(* IEC 61131-3 sources: LStream-JSON-XML/test, 4 files *)

(* ---- JsonDeserializerTests.st ---- *)
USING Simatic.Ax;
USING AxUnit;
USING Simatic.Ax.LStream;
USING Simatic.Ax.LStream.Utilities;
USING Simatic.Ax.System.Strings;
using Simatic.Ax.LStream.Models;

NAMESPACE LStreamTest

    ///////////////// Tests for JSON Blocks
    {TestFixture}
    CLASS JsonDeserializerTests
        VAR
            //Test1 (Test to try the LStream_JsonDeserializer.st by deserializing a JSON (inputString1 & inputString2) and comparing its output with the expected tree (expectedTreeOutput1))
            jsonDeserializer : LStream_JsonDeserializer;
            inputString1 : STRING := '{"sessionContext": {"sessionId": "154237171615905","locale": "en_US","persId": 0},"methodName": "valeo2WC.cfWipClose","inArgs": [{"mode": "0","stationNumber": "SubRib0101","step": "0010","cycleTime": "253.2","unitArray": [';
            inputString2 : STRING := '{"unit": "HLF659734","pos": "1", "state": "1","failArray": [{"failCode": "Condensator position","compName": "BOMPOS60"}]},{"unit": "HLF659735","pos": "2", "state": "0"}]}]}';
            rawInput1 : ARRAY[0..10000] OF BYTE;
            actualTreeOutput : ARRAY[0..200] OF LStream_typeElement;
            expectedTreeOutput1 : ARRAY[0..200] OF LStream_typeElement;

            //Test2 (Test to try the LStream_JsonDeserializer.st when the input JSON has empty brackets as value in the key (In this example: "items":[] & "edges":[]). The deserialize output tree is compared with the expected tree (expectedTreeOutput2))
            jsonDeserializer2 : LStream_JsonDeserializer;
            inputString3 : STRING := '{"id":"A","nodes":[{"nodeId":"CAT","items":[],"sequenceId":"A","released":"WORD","nodePosition":{"x":"1"}}],"edges":[]}';
            rawInput2 : ARRAY[0..10000] OF BYTE;
            actualTreeOutput2 : ARRAY[0..200] OF LStream_typeElement;
            expectedTreeOutput2 : ARRAY[0..200] OF LStream_typeElement;

       END_VAR

        {FixtureSetup}
        METHOD PUBLIC TestSetup

            //Test1 Setup
            StringToByteArray(string1 := inputString1, string2 := inputString2, byteArray := rawInput1);

            expectedTreeOutput1[0].types := SINT#16#0;
            expectedTreeOutput1[0].key := 'sessionContext';
            expectedTreeOutput1[0].value := 'NULL';
            expectedTreeOutput1[0].depth := SINT#16#0;
            expectedTreeOutput1[0].closingElement := FALSE;

            expectedTreeOutput1[1].types := SINT#16#02;
            expectedTreeOutput1[1].key := 'sessionId';
            expectedTreeOutput1[1].value := '154237171615905';
            expectedTreeOutput1[1].depth := SINT#16#01;
            expectedTreeOutput1[1].closingElement := FALSE;

            expectedTreeOutput1[2].types := SINT#16#02;
            expectedTreeOutput1[2].key := 'locale';
            expectedTreeOutput1[2].value := 'en_US';
            expectedTreeOutput1[2].depth := SINT#16#01;
            expectedTreeOutput1[2].closingElement := FALSE;

            expectedTreeOutput1[3].types := SINT#16#03;
            expectedTreeOutput1[3].key := 'persId';
            expectedTreeOutput1[3].value := '0';
            expectedTreeOutput1[3].depth := SINT#16#01;
            expectedTreeOutput1[3].closingElement := TRUE;

            expectedTreeOutput1[4].types := SINT#16#02;
            expectedTreeOutput1[4].key := 'methodName';
            expectedTreeOutput1[4].value := 'valeo2WC.cfWipClose';
            expectedTreeOutput1[4].depth := SINT#16#0;
            expectedTreeOutput1[4].closingElement := FALSE;

            expectedTreeOutput1[5].types := SINT#16#01;
            expectedTreeOutput1[5].key := 'inArgs';
            expectedTreeOutput1[5].value := 'NULL';
            expectedTreeOutput1[5].depth := SINT#16#0;
            expectedTreeOutput1[5].closingElement := false;

            expectedTreeOutput1[6].types := SINT#16#02;
            expectedTreeOutput1[6].key := 'mode';
            expectedTreeOutput1[6].value := '0';
            expectedTreeOutput1[6].depth := SINT#16#02;
            expectedTreeOutput1[6].closingElement := false;

            expectedTreeOutput1[7].types := SINT#16#02;
            expectedTreeOutput1[7].key := 'stationNumber';
            expectedTreeOutput1[7].value := 'SubRib0101';
            expectedTreeOutput1[7].depth := SINT#16#02;
            expectedTreeOutput1[7].closingElement := false;

            expectedTreeOutput1[8].types := SINT#16#02;
            expectedTreeOutput1[8].key := 'step';
            expectedTreeOutput1[8].value := '0010';
            expectedTreeOutput1[8].depth := SINT#16#02;
            expectedTreeOutput1[8].closingElement := false;

            expectedTreeOutput1[9].types := SINT#16#02;
            expectedTreeOutput1[9].key := 'cycleTime';
            expectedTreeOutput1[9].value := '253.2';
            expectedTreeOutput1[9].depth := SINT#16#02;
            expectedTreeOutput1[9].closingElement := false;

            expectedTreeOutput1[10].types := SINT#16#01;
            expectedTreeOutput1[10].key := 'unitArray';
            expectedTreeOutput1[10].value := 'NULL';
            expectedTreeOutput1[10].depth := SINT#16#02;
            expectedTreeOutput1[10].closingElement := false;

            expectedTreeOutput1[11].types := SINT#16#02;
            expectedTreeOutput1[11].key := 'unit';
            expectedTreeOutput1[11].value := 'HLF659734';
            expectedTreeOutput1[11].depth := SINT#16#04;
            expectedTreeOutput1[11].closingElement := false;

            expectedTreeOutput1[12].types := SINT#16#02;
            expectedTreeOutput1[12].key := 'pos';
            expectedTreeOutput1[12].value := '1';
            expectedTreeOutput1[12].depth := SINT#16#04;
            expectedTreeOutput1[12].closingElement := false;

            expectedTreeOutput1[13].types := SINT#16#02;
            expectedTreeOutput1[13].key := 'state';
            expectedTreeOutput1[13].value := '1';
            expectedTreeOutput1[13].depth := SINT#16#04;
            expectedTreeOutput1[13].closingElement := false;

            expectedTreeOutput1[14].types := SINT#16#01;
            expectedTreeOutput1[14].key := 'failArray';
            expectedTreeOutput1[14].value := 'NULL';
            expectedTreeOutput1[14].depth := SINT#16#04;
            expectedTreeOutput1[14].closingElement := false;

            expectedTreeOutput1[15].types := SINT#16#02;
            expectedTreeOutput1[15].key := 'failCode';
            expectedTreeOutput1[15].value := 'Condensator position';
            expectedTreeOutput1[15].depth := SINT#16#06;
            expectedTreeOutput1[15].closingElement := false;

            expectedTreeOutput1[16].types := SINT#16#02;
            expectedTreeOutput1[16].key := 'compName';
            expectedTreeOutput1[16].value := 'BOMPOS60';
            expectedTreeOutput1[16].depth := SINT#16#06;
            expectedTreeOutput1[16].closingElement := true;

            expectedTreeOutput1[17].types := SINT#16#02;
            expectedTreeOutput1[17].key := 'unit';
            expectedTreeOutput1[17].value := 'HLF659735';
            expectedTreeOutput1[17].depth := SINT#16#04;
            expectedTreeOutput1[17].closingElement := FALSE;

            expectedTreeOutput1[18].types := SINT#16#02;
            expectedTreeOutput1[18].key := 'pos';
            expectedTreeOutput1[18].value := '2';
            expectedTreeOutput1[18].depth := SINT#16#04;
            expectedTreeOutput1[18].closingElement := FALSE;

            expectedTreeOutput1[19].types := SINT#16#02;
            expectedTreeOutput1[19].key := 'state';
            expectedTreeOutput1[19].value := '0';
            expectedTreeOutput1[19].depth := SINT#16#04;
            expectedTreeOutput1[19].closingElement := true;

            //Test Setup Json Deserializer case 2
            StringToByteArray(string1 := inputString3, byteArray := rawInput2);

            expectedTreeOutput2[0].types := SINT#16#02;
            expectedTreeOutput2[0].key := 'id';
            expectedTreeOutput2[0].value := 'A';
            expectedTreeOutput2[0].depth := SINT#16#0;
            expectedTreeOutput2[0].closingElement := FALSE;

            expectedTreeOutput2[1].types := SINT#16#01;
            expectedTreeOutput2[1].key := 'nodes';
            expectedTreeOutput2[1].value := 'NULL';
            expectedTreeOutput2[1].depth := SINT#16#0;
            expectedTreeOutput2[1].closingElement := FALSE;

            expectedTreeOutput2[2].types := SINT#16#02;
            expectedTreeOutput2[2].key := 'nodeId';
            expectedTreeOutput2[2].value := 'CAT';
            expectedTreeOutput2[2].depth := SINT#16#02;
            expectedTreeOutput2[2].closingElement := FALSE;

            expectedTreeOutput2[3].types := SINT#16#01;
            expectedTreeOutput2[3].key := 'items';
            expectedTreeOutput2[3].value := 'NULL';
            expectedTreeOutput2[3].depth := SINT#16#02;
            expectedTreeOutput2[3].closingElement := FALSE;

            expectedTreeOutput2[4].types := SINT#16#02;
            expectedTreeOutput2[4].key := 'sequenceId';
            expectedTreeOutput2[4].value := 'A';
            expectedTreeOutput2[4].depth := SINT#16#02;
            expectedTreeOutput2[4].closingElement := FALSE;

            expectedTreeOutput2[5].types := SINT#16#02;
            expectedTreeOutput2[5].key := 'released';
            expectedTreeOutput2[5].value := 'WORD';
            expectedTreeOutput2[5].depth := SINT#16#02;
            expectedTreeOutput2[5].closingElement := FALSE;

            expectedTreeOutput2[6].types := SINT#16#0;
            expectedTreeOutput2[6].key := 'nodePosition';
            expectedTreeOutput2[6].value := 'NULL';
            expectedTreeOutput2[6].depth := SINT#16#02;
            expectedTreeOutput2[6].closingElement := FALSE;

            expectedTreeOutput2[7].types := SINT#16#02;
            expectedTreeOutput2[7].key := 'x';
            expectedTreeOutput2[7].value := '1';
            expectedTreeOutput2[7].depth := SINT#16#03;
            expectedTreeOutput2[7].closingElement := TRUE;

            expectedTreeOutput2[8].types := SINT#16#01;
            expectedTreeOutput2[8].key := 'edges';
            expectedTreeOutput2[8].value := 'NULL';
            expectedTreeOutput2[8].depth := SINT#16#0;
            expectedTreeOutput2[8].closingElement := TRUE;

        END_METHOD

        //Test1
        {Test}
        METHOD PUBLIC TestJsonDeserializer
            VAR
                i : INT;
            END_VAR;
            // Disable timeout timer for the test
            AxUnit.Mocking.Mock(mockeeFn := NAME_OF(System.Timer.OnDelay), mockFn := NAME_OF(Simatic.Ax.Mocks.OnDelayMock_false));

            jsonDeserializer.execute := TRUE;
            WHILE (TRUE) DO
                jsonDeserializer(raw := rawInput1, tree := actualTreeOutput);
                IF(jsonDeserializer.done = TRUE) THEN
                    EXIT;
                END_IF;
                IF(jsonDeserializer.error = TRUE) THEN
                    EXIT;
                END_IF;
            END_WHILE;
            //Tests for block execution
            AxUnit.Assert.Equal(actual := jsonDeserializer.resultCount, expected := 20);
            AXUnit.Assert.Equal(actual := jsonDeserializer.busy, expected := FALSE);
            AXUnit.Assert.Equal(actual := jsonDeserializer.error, expected := FALSE);
            AXUnit.Assert.Equal(actual := jsonDeserializer.done, expected := TRUE);
            AXUnit.Assert.Equal(actual := jsonDeserializer.status, expected := WORD#16#0000);
            //Tests for block output content
            Assert.LStreamTypeElementEqual(actualTreeOutput, expectedTreeOutput1);
        END_METHOD

        //Test2
        {Test}
        METHOD PUBLIC TestJsonDeserializer_EmptyBrackets
            VAR
                i : INT;
            END_VAR;
            // Disable timeout timer for the test
            AxUnit.Mocking.Mock(mockeeFn := NAME_OF(System.Timer.OnDelay), mockFn := NAME_OF(Simatic.Ax.Mocks.OnDelayMock_false));

            jsonDeserializer2.execute := TRUE;
            WHILE (TRUE) DO
                jsonDeserializer2(raw := rawInput2, tree := actualTreeOutput2);
                IF(jsonDeserializer2.done = TRUE) THEN
                    EXIT;
                END_IF;
                IF(jsonDeserializer2.error = TRUE) THEN
                    EXIT;
                END_IF;
            END_WHILE;
            //Tests for block execution
            AxUnit.Assert.Equal(actual := jsonDeserializer2.resultCount, expected := 9);
            AXUnit.Assert.Equal(actual := jsonDeserializer2.busy, expected := FALSE);
            AXUnit.Assert.Equal(actual := jsonDeserializer2.error, expected := FALSE);
            AXUnit.Assert.Equal(actual := jsonDeserializer2.done, expected := TRUE);
            AXUnit.Assert.Equal(actual := jsonDeserializer2.status, expected := WORD#16#0000);
            //Tests for block output content
            Assert.LStreamTypeElementEqual(actualTreeOutput2, expectedTreeOutput2);
        END_METHOD
    END_CLASS

    {TestFixture}
    CLASS JsonDeserializerStatusTest
        VAR
            //Test1 (Test to try the LStream_JsonDeserializer.st by deserializing a JSON (inputString1 & inputString2) and comparing its output with the expected tree (expectedTreeOutput1))
            jsonDeserializer : LStream_JsonDeserializer;
            jsonDeserializerEmpty : LStream_JsonDeserializer;

            // Test Error when given input tree is empty
            rawInputEmpty : ARRAY[0..5] OF BYTE;
            // Test Error when given output tree is empty
            rawInputTreeTooSmall : ARRAY[0..10000] OF BYTE;

            actualTreeOutput : ARRAY[0..0] OF LStream_typeElement;
            actualTreeOutputEmpty : ARRAY[0..0] OF LStream_typeElement;
            inputStringSimple : STRING := '{"id": "A","name":"Too Small Test","year":"2026","sessionContext": {"sessionId":"154237171615905","locale": "en_US","persId": 0}';

        END_VAR

        VAR CONSTANT
            /// No job being currently processed
            STATUS_NO_CALL : Word := WORD#16#7000;
            /// Error: provided array to too small
            ERR_TREE_ARRAY_TOO_SMALL : Word := WORD#16#8201;
            /// Error: no raw data provided
            ERR_EMPTY_RAW_DATA : Word := WORD#16#8401;
            /// Error: due to an undefined state in state machine
            ERR_UNDEFINED_STATE : Word := WORD#16#8600;
        END_VAR

        {TestSetup}
        METHOD PUBLIC TestSetup
            jsonDeserializer := jsonDeserializerEmpty;
            actualTreeOutput := actualTreeOutputEmpty;
        END_METHOD

        {Test}
        METHOD PUBLIC TestJsonDeserializer_ErrorEmptyRawData
            // Disable timeout timer for deterministic parsing progress
            AxUnit.Mocking.Mock(mockeeFn := NAME_OF(System.Timer.OnDelay), mockFn := NAME_OF(Simatic.Ax.Mocks.OnDelayMock_false));

            jsonDeserializer.execute := FALSE;
            jsonDeserializer(raw := rawInputEmpty, tree := actualTreeOutput);

            jsonDeserializer.execute := TRUE;
            WHILE (TRUE) DO
                jsonDeserializer(raw := rawInputEmpty, tree := actualTreeOutput);
                IF(jsonDeserializer.done = TRUE) THEN
                    EXIT;
                END_IF;
                IF(jsonDeserializer.error = TRUE) THEN
                    EXIT;
                END_IF;
            END_WHILE;

            AXUnit.Assert.Equal(actual := jsonDeserializer.done, expected := FALSE);
            AXUnit.Assert.Equal(actual := jsonDeserializer.error, expected := TRUE);
            AXUnit.Assert.Equal(actual := jsonDeserializer.busy, expected := FALSE);
            AXUnit.Assert.Equal(actual := jsonDeserializer.status, expected := ERR_EMPTY_RAW_DATA);

            // Check if error reset
            jsonDeserializer(execute := FALSE, raw := rawInputEmpty, tree := actualTreeOutput);
            AXUnit.Assert.Equal(actual := jsonDeserializer.done, expected := FALSE);
            AXUnit.Assert.Equal(actual := jsonDeserializer.error, expected := FALSE);
            AXUnit.Assert.Equal(actual := jsonDeserializer.busy, expected := FALSE);
            AXUnit.Assert.Equal(actual := jsonDeserializer.status, expected := STATUS_NO_CALL);
        END_METHOD

        {Test}
        METHOD PUBLIC TestJsonDeserializer_ErrorTreeTooSmall
            // Disable timeout timer for deterministic parsing progress
            AxUnit.Mocking.Mock(mockeeFn := NAME_OF(System.Timer.OnDelay), mockFn := NAME_OF(Simatic.Ax.Mocks.OnDelayMock_false));

            // StringToByteArray(string1 := inputStringSimple, byteArray := rawInputTreeTooSmall);
            System.Serialization.Serialize(offset := 0, value := inputStringSimple, buffer := rawInputTreeTooSmall);

            jsonDeserializer.execute := FALSE;
            jsonDeserializer(raw := rawInputTreeTooSmall, tree := actualTreeOutput);

            jsonDeserializer.execute := TRUE;
            WHILE (TRUE) DO
                jsonDeserializer(raw := rawInputTreeTooSmall, tree := actualTreeOutput);
                IF(jsonDeserializer.done = TRUE) THEN
                    EXIT;
                END_IF;
                IF(jsonDeserializer.error = TRUE) THEN
                    EXIT;
                END_IF;
            END_WHILE;

            AXUnit.Assert.Equal(actual := jsonDeserializer.done, expected := FALSE);
            AXUnit.Assert.Equal(actual := jsonDeserializer.error, expected := TRUE);
            AXUnit.Assert.Equal(actual := jsonDeserializer.busy, expected := FALSE);
            AXUnit.Assert.Equal(actual := jsonDeserializer.status, expected := ERR_TREE_ARRAY_TOO_SMALL);

            // Check if error reset
            jsonDeserializer(execute := FALSE, raw := rawInputTreeTooSmall, tree := actualTreeOutput);
            AXUnit.Assert.Equal(actual := jsonDeserializer.done, expected := FALSE);
            AXUnit.Assert.Equal(actual := jsonDeserializer.error, expected := FALSE);
            AXUnit.Assert.Equal(actual := jsonDeserializer.busy, expected := FALSE);
            AXUnit.Assert.Equal(actual := jsonDeserializer.status, expected := STATUS_NO_CALL);
        END_METHOD
    END_CLASS
END_NAMESPACE

(* ---- JsonSerializerTests.st ---- *)
USING Simatic.Ax;
USING AxUnit;
USING Simatic.Ax.LStream;
USING Simatic.Ax.LStream.Utilities;
USING System.Strings;
using Simatic.Ax.LStream.Models;
using System.Serialization;

NAMESPACE LStreamTest

    {TestFixture}
    CLASS JsonSerializerTests
        VAR

            //Test1 (Test to try the LStream_JsonSerializer.st by serializing a tree (treeInput) and comparing its output with the expected byte array (expectedJsonByteOutputResult))
            jsonSerializer : LStream_JsonSerializer;
            jsonByteOutputResult : ARRAY[0..600] OF BYTE;
            treeInput : ARRAY[0..200] OF LStream_typeElement;
            expectedJsonByteOutputResult : ARRAY[0..600] OF BYTE := [
            BYTE#16#7B, BYTE#16#22, BYTE#16#73, BYTE#16#65, BYTE#16#73, BYTE#16#73, BYTE#16#69, BYTE#16#6F, BYTE#16#6E, BYTE#16#43, BYTE#16#6F, BYTE#16#6E, BYTE#16#74, BYTE#16#65, BYTE#16#78, BYTE#16#74, BYTE#16#22, BYTE#16#3A, BYTE#16#7B, BYTE#16#22, BYTE#16#73, BYTE#16#65, BYTE#16#73, BYTE#16#73, BYTE#16#69, BYTE#16#6F, BYTE#16#6E, BYTE#16#49, BYTE#16#64, BYTE#16#22, BYTE#16#3A, BYTE#16#22, BYTE#16#31, BYTE#16#35, BYTE#16#34, BYTE#16#32, BYTE#16#33, BYTE#16#37, BYTE#16#31, BYTE#16#37, BYTE#16#31, BYTE#16#36, BYTE#16#31, BYTE#16#35, BYTE#16#39, BYTE#16#30, BYTE#16#35, BYTE#16#22, BYTE#16#2C, BYTE#16#22, BYTE#16#6C, BYTE#16#6F, BYTE#16#63, BYTE#16#61, BYTE#16#6C, BYTE#16#65, BYTE#16#22, BYTE#16#3A, BYTE#16#22, BYTE#16#65, BYTE#16#6E, BYTE#16#5F, BYTE#16#55, BYTE#16#53, BYTE#16#22, BYTE#16#2C, BYTE#16#22, BYTE#16#70, BYTE#16#65, BYTE#16#72, BYTE#16#73, BYTE#16#49, BYTE#16#64, BYTE#16#22, BYTE#16#3A, BYTE#16#30, BYTE#16#7D, BYTE#16#2C, BYTE#16#22, BYTE#16#6D, BYTE#16#65, BYTE#16#74, BYTE#16#68, BYTE#16#6F, BYTE#16#64, BYTE#16#4E, BYTE#16#61, BYTE#16#6D, BYTE#16#65, BYTE#16#22, BYTE#16#3A, BYTE#16#22, BYTE#16#76, BYTE#16#61, BYTE#16#6C, BYTE#16#65, BYTE#16#6F, BYTE#16#32, BYTE#16#57, BYTE#16#43, BYTE#16#2E, BYTE#16#63, BYTE#16#66, BYTE#16#57, BYTE#16#69, BYTE#16#70, BYTE#16#43, BYTE#16#6C, BYTE#16#6F, BYTE#16#73, BYTE#16#65, BYTE#16#22, BYTE#16#2C, BYTE#16#22, BYTE#16#69, BYTE#16#6E, BYTE#16#41, BYTE#16#72, BYTE#16#67, BYTE#16#73, BYTE#16#22, BYTE#16#3A, BYTE#16#5B, BYTE#16#7B, BYTE#16#22, BYTE#16#6D, BYTE#16#6F, BYTE#16#64, BYTE#16#65, BYTE#16#22, BYTE#16#3A, BYTE#16#22, BYTE#16#30, BYTE#16#22, BYTE#16#2C, BYTE#16#22, BYTE#16#73, BYTE#16#74, BYTE#16#61, BYTE#16#74, BYTE#16#69, BYTE#16#6F, BYTE#16#6E, BYTE#16#4E, BYTE#16#75, BYTE#16#6D, BYTE#16#62, BYTE#16#65, BYTE#16#72, BYTE#16#22, BYTE#16#3A, BYTE#16#22, BYTE#16#53, BYTE#16#75, BYTE#16#62, BYTE#16#52, BYTE#16#69, BYTE#16#62, BYTE#16#30, BYTE#16#31, BYTE#16#30, BYTE#16#31, BYTE#16#22, BYTE#16#2C, BYTE#16#22, BYTE#16#73, BYTE#16#74, BYTE#16#65, BYTE#16#70, BYTE#16#22, BYTE#16#3A, BYTE#16#22, BYTE#16#30, BYTE#16#30, BYTE#16#31, BYTE#16#30, BYTE#16#22, BYTE#16#2C, BYTE#16#22, BYTE#16#63, BYTE#16#79, BYTE#16#63, BYTE#16#6C, BYTE#16#65, BYTE#16#54, BYTE#16#69, BYTE#16#6D, BYTE#16#65, BYTE#16#22, BYTE#16#3A, BYTE#16#22, BYTE#16#32, BYTE#16#35, BYTE#16#33, BYTE#16#2E, BYTE#16#32, BYTE#16#22, BYTE#16#2C, BYTE#16#22, BYTE#16#75, BYTE#16#6E, BYTE#16#69, BYTE#16#74, BYTE#16#41, BYTE#16#72, BYTE#16#72, BYTE#16#61, BYTE#16#79, BYTE#16#22, BYTE#16#3A, BYTE#16#5B, BYTE#16#7B, BYTE#16#22, BYTE#16#75, BYTE#16#6E, BYTE#16#69, BYTE#16#74, BYTE#16#22, BYTE#16#3A, BYTE#16#22, BYTE#16#48, BYTE#16#4C, BYTE#16#46, BYTE#16#36, BYTE#16#35, BYTE#16#39, BYTE#16#37, BYTE#16#33, BYTE#16#34, BYTE#16#22, BYTE#16#2C, BYTE#16#22, BYTE#16#70, BYTE#16#6F, BYTE#16#73, BYTE#16#22, BYTE#16#3A, BYTE#16#22, BYTE#16#31, BYTE#16#22, BYTE#16#2C, BYTE#16#22, BYTE#16#73, BYTE#16#74, BYTE#16#61, BYTE#16#74, BYTE#16#65, BYTE#16#22, BYTE#16#3A, BYTE#16#22, BYTE#16#31, BYTE#16#22, BYTE#16#2C, BYTE#16#22, BYTE#16#66, BYTE#16#61, BYTE#16#69, BYTE#16#6C, BYTE#16#41, BYTE#16#72, BYTE#16#72, BYTE#16#61, BYTE#16#79, BYTE#16#22, BYTE#16#3A, BYTE#16#5B, BYTE#16#7B, BYTE#16#22, BYTE#16#66, BYTE#16#61, BYTE#16#69, BYTE#16#6C, BYTE#16#43, BYTE#16#6F, BYTE#16#64, BYTE#16#65, BYTE#16#22, BYTE#16#3A, BYTE#16#22, BYTE#16#43, BYTE#16#6F, BYTE#16#6E, BYTE#16#64, BYTE#16#65, BYTE#16#6E, BYTE#16#73, BYTE#16#61, BYTE#16#74, BYTE#16#6F, BYTE#16#72, BYTE#16#20, BYTE#16#70, BYTE#16#6F, BYTE#16#73, BYTE#16#69, BYTE#16#74, BYTE#16#69, BYTE#16#6F, BYTE#16#6E, BYTE#16#22, BYTE#16#2C, BYTE#16#22, BYTE#16#63, BYTE#16#6F, BYTE#16#6D, BYTE#16#70, BYTE#16#4E, BYTE#16#61, BYTE#16#6D, BYTE#16#65, BYTE#16#22, BYTE#16#3A, BYTE#16#22, BYTE#16#42, BYTE#16#4F, BYTE#16#4D, BYTE#16#50, BYTE#16#4F, BYTE#16#53, BYTE#16#36, BYTE#16#30, BYTE#16#22, BYTE#16#7D, BYTE#16#5D, BYTE#16#2C, BYTE#16#22, BYTE#16#75, BYTE#16#6E, BYTE#16#69, BYTE#16#74, BYTE#16#22, BYTE#16#3A, BYTE#16#22, BYTE#16#48, BYTE#16#4C, BYTE#16#46, BYTE#16#36, BYTE#16#35, BYTE#16#39, BYTE#16#37, BYTE#16#33, BYTE#16#35, BYTE#16#22, BYTE#16#2C, BYTE#16#22, BYTE#16#70, BYTE#16#6F, BYTE#16#73, BYTE#16#22, BYTE#16#3A, BYTE#16#22, BYTE#16#32, BYTE#16#22, BYTE#16#2C, BYTE#16#22, BYTE#16#73, BYTE#16#74, BYTE#16#61, BYTE#16#74, BYTE#16#65, BYTE#16#22, BYTE#16#3A, BYTE#16#22, BYTE#16#30, BYTE#16#22, BYTE#16#7D, BYTE#16#5D, BYTE#16#7D, BYTE#16#5D, BYTE#16#7D,
            BYTE#16#0, BYTE#16#0, BYTE#16#0, BYTE#16#0, BYTE#16#0, BYTE#16#0, BYTE#16#0, BYTE#16#0, BYTE#16#0, BYTE#16#0,
            BYTE#16#0, BYTE#16#0, BYTE#16#0, BYTE#16#0, BYTE#16#0, BYTE#16#0, BYTE#16#0, BYTE#16#0, BYTE#16#0, BYTE#16#0,
            BYTE#16#0, BYTE#16#0, BYTE#16#0, BYTE#16#0, BYTE#16#0, BYTE#16#0, BYTE#16#0, BYTE#16#0, BYTE#16#0, BYTE#16#0,
            BYTE#16#0, BYTE#16#0, BYTE#16#0, BYTE#16#0, BYTE#16#0, BYTE#16#0, BYTE#16#0, BYTE#16#0, BYTE#16#0, BYTE#16#0,
            BYTE#16#0, BYTE#16#0, BYTE#16#0, BYTE#16#0, BYTE#16#0, BYTE#16#0, BYTE#16#0, BYTE#16#0, BYTE#16#0, BYTE#16#0,
            BYTE#16#0, BYTE#16#0, BYTE#16#0, BYTE#16#0, BYTE#16#0, BYTE#16#0, BYTE#16#0, BYTE#16#0, BYTE#16#0, BYTE#16#0,
            BYTE#16#0, BYTE#16#0, BYTE#16#0, BYTE#16#0, BYTE#16#0, BYTE#16#0, BYTE#16#0, BYTE#16#0, BYTE#16#0, BYTE#16#0,
            BYTE#16#0, BYTE#16#0, BYTE#16#0, BYTE#16#0, BYTE#16#0, BYTE#16#0, BYTE#16#0, BYTE#16#0, BYTE#16#0, BYTE#16#0,
            BYTE#16#0, BYTE#16#0, BYTE#16#0, BYTE#16#0, BYTE#16#0, BYTE#16#0, BYTE#16#0, BYTE#16#0, BYTE#16#0, BYTE#16#0,
            BYTE#16#0, BYTE#16#0, BYTE#16#0, BYTE#16#0, BYTE#16#0, BYTE#16#0, BYTE#16#0, BYTE#16#0, BYTE#16#0, BYTE#16#0,
            BYTE#16#0, BYTE#16#0, BYTE#16#0, BYTE#16#0, BYTE#16#0, BYTE#16#0, BYTE#16#0, BYTE#16#0, BYTE#16#0, BYTE#16#0,
            BYTE#16#0, BYTE#16#0, BYTE#16#0, BYTE#16#0, BYTE#16#0, BYTE#16#0, BYTE#16#0, BYTE#16#0, BYTE#16#0, BYTE#16#0,
            BYTE#16#0, BYTE#16#0, BYTE#16#0, BYTE#16#0, BYTE#16#0, BYTE#16#0, BYTE#16#0, BYTE#16#0, BYTE#16#0, BYTE#16#0,
            BYTE#16#0, BYTE#16#0, BYTE#16#0, BYTE#16#0, BYTE#16#0, BYTE#16#0, BYTE#16#0, BYTE#16#0, BYTE#16#0, BYTE#16#0,
            BYTE#16#0, BYTE#16#0, BYTE#16#0, BYTE#16#0, BYTE#16#0, BYTE#16#0, BYTE#16#0, BYTE#16#0, BYTE#16#0, BYTE#16#0,
            BYTE#16#0, BYTE#16#0, BYTE#16#0, BYTE#16#0, BYTE#16#0, BYTE#16#0, BYTE#16#0, BYTE#16#0, BYTE#16#0, BYTE#16#0,
            BYTE#16#0, BYTE#16#0, BYTE#16#0, BYTE#16#0, BYTE#16#0, BYTE#16#0, BYTE#16#0, BYTE#16#0, BYTE#16#0, BYTE#16#0,
            BYTE#16#0, BYTE#16#0, BYTE#16#0, BYTE#16#0, BYTE#16#0, BYTE#16#0, BYTE#16#0, BYTE#16#0, BYTE#16#0, BYTE#16#0,
            BYTE#16#0, BYTE#16#0, BYTE#16#0, BYTE#16#0, BYTE#16#0, BYTE#16#0, BYTE#16#0, BYTE#16#0, BYTE#16#0, BYTE#16#0,
            BYTE#16#0, BYTE#16#0, BYTE#16#0, BYTE#16#0, BYTE#16#0, BYTE#16#0, BYTE#16#0, BYTE#16#0, BYTE#16#0, BYTE#16#0,
            BYTE#16#0, BYTE#16#0, BYTE#16#0, BYTE#16#0, BYTE#16#0, BYTE#16#0, BYTE#16#0, BYTE#16#0, BYTE#16#0, BYTE#16#0,
            BYTE#16#0, BYTE#16#0, BYTE#16#0, BYTE#16#0, BYTE#16#0, BYTE#16#0, BYTE#16#0, BYTE#16#0, BYTE#16#0, BYTE#16#0,
            BYTE#16#0, BYTE#16#0, BYTE#16#0, BYTE#16#0, BYTE#16#0, BYTE#16#0, BYTE#16#0, BYTE#16#0, BYTE#16#0, BYTE#16#0,
            BYTE#16#0
];

            //Test2 (Test to try the LStream_JsonSerializer.st when the input tree (treeInput2) has empty arrays (treeInput2[8] & treeInput2[3]) nodes (Coming from a JSON with empty brackets [] in its structure))
            jsonSerializer2 : LStream_JsonSerializer;
            jsonByteOutputResult2 : ARRAY[0..600] OF BYTE;
            treeInput2 : ARRAY[0..200] OF LStream_typeElement;
            expectedJsonByteOutputResult2 : ARRAY[0..119] OF BYTE := [
            BYTE#16#7B, BYTE#16#22, BYTE#16#69, BYTE#16#64, BYTE#16#22, BYTE#16#3A, BYTE#16#22, BYTE#16#41, BYTE#16#22, BYTE#16#2C,
            BYTE#16#22, BYTE#16#6E, BYTE#16#6F, BYTE#16#64, BYTE#16#65, BYTE#16#73, BYTE#16#22, BYTE#16#3A, BYTE#16#5B, BYTE#16#7B,
            BYTE#16#22, BYTE#16#6E, BYTE#16#6F, BYTE#16#64, BYTE#16#65, BYTE#16#49, BYTE#16#64, BYTE#16#22, BYTE#16#3A, BYTE#16#22,
            BYTE#16#43, BYTE#16#41, BYTE#16#54, BYTE#16#22, BYTE#16#2C, BYTE#16#22, BYTE#16#69, BYTE#16#74, BYTE#16#65, BYTE#16#6D,
            BYTE#16#73, BYTE#16#22, BYTE#16#3A, BYTE#16#5B, BYTE#16#5D, BYTE#16#2C, BYTE#16#22, BYTE#16#73, BYTE#16#65, BYTE#16#71,
            BYTE#16#75, BYTE#16#65, BYTE#16#6E, BYTE#16#63, BYTE#16#65, BYTE#16#49, BYTE#16#64, BYTE#16#22, BYTE#16#3A, BYTE#16#22,
            BYTE#16#41, BYTE#16#22, BYTE#16#2C, BYTE#16#22, BYTE#16#72, BYTE#16#65, BYTE#16#6C, BYTE#16#65, BYTE#16#61, BYTE#16#73,
            BYTE#16#65, BYTE#16#64, BYTE#16#22, BYTE#16#3A, BYTE#16#22, BYTE#16#57, BYTE#16#4F, BYTE#16#52, BYTE#16#44, BYTE#16#22,
            BYTE#16#2C, BYTE#16#22, BYTE#16#6E, BYTE#16#6F, BYTE#16#64, BYTE#16#65, BYTE#16#50, BYTE#16#6F, BYTE#16#73, BYTE#16#69,
            BYTE#16#74, BYTE#16#69, BYTE#16#6F, BYTE#16#6E, BYTE#16#22, BYTE#16#3A, BYTE#16#7B, BYTE#16#22, BYTE#16#78, BYTE#16#22,
            BYTE#16#3A, BYTE#16#22, BYTE#16#31, BYTE#16#22, BYTE#16#7D, BYTE#16#7D, BYTE#16#5D, BYTE#16#2C, BYTE#16#22, BYTE#16#65,
            BYTE#16#64, BYTE#16#67, BYTE#16#65, BYTE#16#73, BYTE#16#22, BYTE#16#3A, BYTE#16#5B, BYTE#16#5D, BYTE#16#7D, BYTE#16#00
];

        END_VAR

        {FixtureSetup}
        METHOD PUBLIC TestSetup
            //Test1 Setup
            //Populate expected LStreamTypeElementArray
            //Populate expectedTreeOutput
                treeInput[0].types := SINT#16#0;
                treeInput[0].key := 'sessionContext';
                treeInput[0].value := 'NULL';
                treeInput[0].depth := SINT#16#0;
                treeInput[0].closingElement := FALSE;

                treeInput[1].types := SINT#16#02;
                treeInput[1].key := 'sessionId';
                treeInput[1].value := '154237171615905';
                treeInput[1].depth := SINT#16#01;
                treeInput[1].closingElement := FALSE;

                treeInput[2].types := SINT#16#02;
                treeInput[2].key := 'locale';
                treeInput[2].value := 'en_US';
                treeInput[2].depth := SINT#16#01;
                treeInput[2].closingElement := FALSE;

                treeInput[3].types := SINT#16#03;
                treeInput[3].key := 'persId';
                treeInput[3].value := '0';
                treeInput[3].depth := SINT#16#01;
                treeInput[3].closingElement := TRUE;

                treeInput[4].types := SINT#16#02;
                treeInput[4].key := 'methodName';
                treeInput[4].value := 'valeo2WC.cfWipClose';
                treeInput[4].depth := SINT#16#0;
                treeInput[4].closingElement := FALSE;

                treeInput[5].types := SINT#16#01;
                treeInput[5].key := 'inArgs';
                treeInput[5].value := 'NULL';
                treeInput[5].depth := SINT#16#0;
                treeInput[5].closingElement := false;

                treeInput[6].types := SINT#16#02;
                treeInput[6].key := 'mode';
                treeInput[6].value := '0';
                treeInput[6].depth := SINT#16#02;
                treeInput[6].closingElement := false;

                treeInput[7].types := SINT#16#02;
                treeInput[7].key := 'stationNumber';
                treeInput[7].value := 'SubRib0101';
                treeInput[7].depth := SINT#16#02;
                treeInput[7].closingElement := false;

                treeInput[8].types := SINT#16#02;
                treeInput[8].key := 'step';
                treeInput[8].value := '0010';
                treeInput[8].depth := SINT#16#02;
                treeInput[8].closingElement := false;

                treeInput[9].types := SINT#16#02;
                treeInput[9].key := 'cycleTime';
                treeInput[9].value := '253.2';
                treeInput[9].depth := SINT#16#02;
                treeInput[9].closingElement := false;

                treeInput[10].types := SINT#16#01;
                treeInput[10].key := 'unitArray';
                treeInput[10].value := 'NULL';
                treeInput[10].depth := SINT#16#02;
                treeInput[10].closingElement := false;

                treeInput[11].types := SINT#16#02;
                treeInput[11].key := 'unit';
                treeInput[11].value := 'HLF659734';
                treeInput[11].depth := SINT#16#04;
                treeInput[11].closingElement := false;

                treeInput[12].types := SINT#16#02;
                treeInput[12].key := 'pos';
                treeInput[12].value := '1';
                treeInput[12].depth := SINT#16#04;
                treeInput[12].closingElement := false;

                treeInput[13].types := SINT#16#02;
                treeInput[13].key := 'state';
                treeInput[13].value := '1';
                treeInput[13].depth := SINT#16#04;
                treeInput[13].closingElement := false;

                treeInput[14].types := SINT#16#01;
                treeInput[14].key := 'failArray';
                treeInput[14].value := 'NULL';
                treeInput[14].depth := SINT#16#04;
                treeInput[14].closingElement := false;

                treeInput[15].types := SINT#16#02;
                treeInput[15].key := 'failCode';
                treeInput[15].value := 'Condensator position';
                treeInput[15].depth := SINT#16#06;
                treeInput[15].closingElement := false;

                treeInput[16].types := SINT#16#02;
                treeInput[16].key := 'compName';
                treeInput[16].value := 'BOMPOS60';
                treeInput[16].depth := SINT#16#06;
                treeInput[16].closingElement := true;

                treeInput[17].types := SINT#16#02;
                treeInput[17].key := 'unit';
                treeInput[17].value := 'HLF659735';
                treeInput[17].depth := SINT#16#04;
                treeInput[17].closingElement := FALSE;

                treeInput[18].types := SINT#16#02;
                treeInput[18].key := 'pos';
                treeInput[18].value := '2';
                treeInput[18].depth := SINT#16#04;
                treeInput[18].closingElement := FALSE;

                treeInput[19].types := SINT#16#02;
                treeInput[19].key := 'state';
                treeInput[19].value := '0';
                treeInput[19].depth := SINT#16#04;
                treeInput[19].closingElement := true;

            //Test2 Setup
            //Populate expected LStreamTypeElementArray
            //Populate expectedTreeOutput
                treeInput2[0].types := SINT#16#02;
                treeInput2[0].key := 'id';
                treeInput2[0].value := 'A';
                treeInput2[0].depth := SINT#16#0;
                treeInput2[0].closingElement := FALSE;

                treeInput2[1].types := SINT#16#01;
                treeInput2[1].key := 'nodes';
                treeInput2[1].value := 'NULL';
                treeInput2[1].depth := SINT#16#0;
                treeInput2[1].closingElement := FALSE;

                treeInput2[2].types := SINT#16#02;
                treeInput2[2].key := 'nodeId';
                treeInput2[2].value := 'CAT';
                treeInput2[2].depth := SINT#16#02;
                treeInput2[2].closingElement := FALSE;

                treeInput2[3].types := SINT#16#01;
                treeInput2[3].key := 'items';
                treeInput2[3].value := 'NULL';
                treeInput2[3].depth := SINT#16#02;
                treeInput2[3].closingElement := FALSE;

                treeInput2[4].types := SINT#16#02;
                treeInput2[4].key := 'sequenceId';
                treeInput2[4].value := 'A';
                treeInput2[4].depth := SINT#16#02;
                treeInput2[4].closingElement := FALSE;

                treeInput2[5].types := SINT#16#02;
                treeInput2[5].key := 'released';
                treeInput2[5].value := 'WORD';
                treeInput2[5].depth := SINT#16#02;
                treeInput2[5].closingElement := FALSE;

                treeInput2[6].types := SINT#16#0;
                treeInput2[6].key := 'nodePosition';
                treeInput2[6].value := 'NULL';
                treeInput2[6].depth := SINT#16#02;
                treeInput2[6].closingElement := FALSE;

                treeInput2[7].types := SINT#16#02;
                treeInput2[7].key := 'x';
                treeInput2[7].value := '1';
                treeInput2[7].depth := SINT#16#03;
                treeInput2[7].closingElement := TRUE;

                treeInput2[8].types := SINT#16#01;
                treeInput2[8].key := 'edges';
                treeInput2[8].value := 'NULL';
                treeInput2[8].depth := SINT#16#0;
                treeInput2[8].closingElement := TRUE;
        END_METHOD

        //Test1
        {Test}
        METHOD PUBLIC TestJsonSerializer
            VAR
                i : INT;
            END_VAR;
            // Disable timeout timer for the test
            AxUnit.Mocking.Mock(mockeeFn := NAME_OF(System.Timer.OnDelay), mockFn := NAME_OF(Simatic.Ax.Mocks.OnDelayMock_false));

            jsonSerializer.execute := TRUE;
            WHILE (TRUE) DO
                jsonSerializer(tree := treeInput, jsonByteArray := jsonByteOutputResult);
                IF(jsonSerializer.done = TRUE) THEN
                    EXIT;
                END_IF;
                IF(jsonSerializer.error = TRUE) THEN
                    EXIT;
                END_IF;
            END_WHILE;
            //Test block execution
            AxUnit.Assert.Equal(actual := jsonSerializer.count, expected := UINT#370);
            AXUnit.Assert.Equal(actual := jsonSerializer.busy, expected := FALSE);
            AXUnit.Assert.Equal(actual := jsonSerializer.error, expected := FALSE);
            AXUnit.Assert.Equal(actual := jsonSerializer.done, expected := TRUE);
            //Test Output Content
            FOR i := 0 TO 400 DO
                AxUnit.Assert.Equal(jsonByteOutputResult[i], expectedJsonByteOutputResult[i]);

            END_FOR;
        END_METHOD

        //Test2
        {Test}
        METHOD PUBLIC TestJsonSerializer_EmptyBrackets
            VAR
                i : INT;
            END_VAR;
            // Disable timeout timer for the test
            AxUnit.Mocking.Mock(mockeeFn := NAME_OF(System.Timer.OnDelay), mockFn := NAME_OF(Simatic.Ax.Mocks.OnDelayMock_false));

            jsonSerializer2.execute := TRUE;
            WHILE (TRUE) DO
                jsonSerializer2(tree := treeInput2, jsonByteArray := jsonByteOutputResult2);
                IF(jsonSerializer2.done = TRUE) THEN
                    EXIT;
                END_IF;
                IF(jsonSerializer2.error = TRUE) THEN
                    EXIT;
                END_IF;
            END_WHILE;
            //Test block execution
            AxUnit.Assert.Equal(actual := jsonSerializer2.count, expected := UINT#119);
            AXUnit.Assert.Equal(actual := jsonSerializer2.busy, expected := FALSE);
            AXUnit.Assert.Equal(actual := jsonSerializer2.error, expected := FALSE);
            AXUnit.Assert.Equal(actual := jsonSerializer2.done, expected := TRUE);
            //Test Output Content
            FOR i := 0 TO 119 DO
                AxUnit.Assert.Equal(jsonByteOutputResult2[i], expectedJsonByteOutputResult2[i]);

            END_FOR;
        END_METHOD
    END_CLASS
END_NAMESPACE

(* ---- XmlDeserializerTests.st ---- *)
USING Simatic;
USING AxUnit;
USING Simatic.Ax.LStream;
USING Simatic.Ax.LStream.Utilities;
USING System.Strings;
USING Simatic.Ax.LStream.Models;

NAMESPACE LStreamTest
    ///////////////// Tests for XML Blocks
    {TestFixture}
    CLASS XmlDeserializerTests
        VAR
            //Test1 (Test to try the LStream_XmlDeserializer.st by deserializing XML (rawInput1, rawInput2, rawInput3) and comparing its output with the expected tree (expectedTreeOutput1))
            xmlDeserializer : LStream_XmlDeserializer;
            rawInput : ARRAY[0..10000] OF BYTE;
            actualTreeOutput : ARRAY[0..200] OF LStream_typeElement;
            expectedTreeOutput1 : ARRAY[0..200] OF LStream_typeElement;

            rawInput1 : STRING := '<?xml version="1.0" encoding="ASCII"?><bookstore><book category="Fiction"><title lang="en">The Great Gatsby</title><author>F. Scott Fitzgerald</author><year>1925</year>';
            rawInput2 : STRING := '<price>10.99</price></book><book category="Programming"><title lang="en">Learning XML</title><author>Erik T. Ray</author><year>2003</year><price>39.95</price></book>';
            rawInput3 : STRING := '<book category="Fantasy"><title lang="en">Harry Potter and the Philosophers Stone</title><author>J.K. Rowling</author><year>1997</year><price>20.00</price></book></bookstore>';

            //Test2 (Test to try the LStream_XmlDeserializer.st when the input XML has spaces before the equals sign in attributes (category = "Science Fiction" or lang   ="en").
            //The deserialize output tree is compared with the expected tree (expectedTreeOutput2))
            xmlDeserializer2 : LStream_XmlDeserializer;
            rawInput4 : STRING := '<bookstore><book category = "Science Fiction" lang   ="en"><title>The Great Gatsby</title><author>F. Scott Fitzgerald</author><year>1925</year><price>10.99</price></book></bookstore>';
            rawInput_2 : ARRAY[0..10000] OF BYTE;
            actualTreeOutput2 : ARRAY[0..200] OF LStream_typeElement;
            expectedTreeOutput2 : ARRAY[0..200] OF LStream_typeElement;

        END_VAR

        {TestSetup}
        METHOD PUBLIC TestSetup
            // Disable timeout timer for all tests
            AxUnit.Mocking.Mock(mockeeFn := NAME_OF(System.Timer.OnDelay), mockFn := NAME_OF(Simatic.Ax.Mocks.OnDelayMock_false));
            //Init timer and expected outputs
            expectedTreeOutput1[0].types := SINT#16#0;
            expectedTreeOutput1[0].key := 'bookstore';
            expectedTreeOutput1[0].value := 'NULL';
            expectedTreeOutput1[0].depth := SINT#16#01;
            expectedTreeOutput1[0].closingElement := FALSE;

            expectedTreeOutput1[1].types := SINT#16#0;
            expectedTreeOutput1[1].key := 'book';
            expectedTreeOutput1[1].value := 'NULL';
            expectedTreeOutput1[1].depth := SINT#16#02;
            expectedTreeOutput1[1].closingElement := FALSE;

            expectedTreeOutput1[2].types := SINT#16#01;
            expectedTreeOutput1[2].key := 'category';
            expectedTreeOutput1[2].value := 'Fiction';
            expectedTreeOutput1[2].depth := SINT#16#02;
            expectedTreeOutput1[2].closingElement := FALSE;

            expectedTreeOutput1[3].types := SINT#16#0;
            expectedTreeOutput1[3].key := 'title';
            expectedTreeOutput1[3].value := 'The Great Gatsby';
            expectedTreeOutput1[3].depth := SINT#16#03;
            expectedTreeOutput1[3].closingElement := FALSE;

            expectedTreeOutput1[4].types := SINT#16#01;
            expectedTreeOutput1[4].key := 'lang';
            expectedTreeOutput1[4].value := 'en';
            expectedTreeOutput1[4].depth := SINT#16#03;
            expectedTreeOutput1[4].closingElement := FALSE;

            expectedTreeOutput1[5].types := SINT#16#0;
            expectedTreeOutput1[5].key := 'author';
            expectedTreeOutput1[5].value := 'F. Scott Fitzgerald';
            expectedTreeOutput1[5].depth := SINT#16#03;
            expectedTreeOutput1[5].closingElement := false;

            expectedTreeOutput1[6].types := SINT#16#0;
            expectedTreeOutput1[6].key := 'year';
            expectedTreeOutput1[6].value := '1925';
            expectedTreeOutput1[6].depth := SINT#16#03;
            expectedTreeOutput1[6].closingElement := false;

            expectedTreeOutput1[7].types := SINT#16#0;
            expectedTreeOutput1[7].key := 'price';
            expectedTreeOutput1[7].value := '10.99';
            expectedTreeOutput1[7].depth := SINT#16#03;
            expectedTreeOutput1[7].closingElement := false;

            expectedTreeOutput1[8].types := SINT#16#0;
            expectedTreeOutput1[8].key := 'book';
            expectedTreeOutput1[8].value := 'NULL';
            expectedTreeOutput1[8].depth := SINT#16#02;
            expectedTreeOutput1[8].closingElement := false;

            expectedTreeOutput1[9].types := SINT#16#01;
            expectedTreeOutput1[9].key := 'category';
            expectedTreeOutput1[9].value := 'Programming';
            expectedTreeOutput1[9].depth := SINT#16#02;
            expectedTreeOutput1[9].closingElement := false;

            expectedTreeOutput1[10].types := SINT#16#0;
            expectedTreeOutput1[10].key := 'title';
            expectedTreeOutput1[10].value := 'Learning XML';
            expectedTreeOutput1[10].depth := SINT#16#03;
            expectedTreeOutput1[10].closingElement := false;

            expectedTreeOutput1[11].types := SINT#16#01;
            expectedTreeOutput1[11].key := 'lang';
            expectedTreeOutput1[11].value := 'en';
            expectedTreeOutput1[11].depth := SINT#16#03;
            expectedTreeOutput1[11].closingElement := FALSE;

            expectedTreeOutput1[12].types := SINT#16#0;
            expectedTreeOutput1[12].key := 'author';
            expectedTreeOutput1[12].value := 'Erik T. Ray';
            expectedTreeOutput1[12].depth := SINT#16#03;
            expectedTreeOutput1[12].closingElement := false;

            expectedTreeOutput1[13].types := SINT#16#0;
            expectedTreeOutput1[13].key := 'year';
            expectedTreeOutput1[13].value := '2003';
            expectedTreeOutput1[13].depth := SINT#16#03;
            expectedTreeOutput1[13].closingElement := false;

            expectedTreeOutput1[14].types := SINT#16#0;
            expectedTreeOutput1[14].key := 'price';
            expectedTreeOutput1[14].value := '39.95';
            expectedTreeOutput1[14].depth := SINT#16#03;
            expectedTreeOutput1[14].closingElement := false;

            expectedTreeOutput1[15].types := SINT#16#0;
            expectedTreeOutput1[15].key := 'book';
            expectedTreeOutput1[15].value := 'NULL';
            expectedTreeOutput1[15].depth := SINT#16#02;
            expectedTreeOutput1[15].closingElement := false;

            expectedTreeOutput1[16].types := SINT#16#01;
            expectedTreeOutput1[16].key := 'category';
            expectedTreeOutput1[16].value := 'Fantasy';
            expectedTreeOutput1[16].depth := SINT#16#02;
            expectedTreeOutput1[16].closingElement := FALSE;

            expectedTreeOutput1[17].types := SINT#16#0;
            expectedTreeOutput1[17].key := 'title';
            expectedTreeOutput1[17].value := 'Harry Potter and the Philosophers Stone';
            expectedTreeOutput1[17].depth := SINT#16#03;
            expectedTreeOutput1[17].closingElement := FALSE;

            expectedTreeOutput1[18].types := SINT#16#01;
            expectedTreeOutput1[18].key := 'lang';
            expectedTreeOutput1[18].value := 'en';
            expectedTreeOutput1[18].depth := SINT#16#03;
            expectedTreeOutput1[18].closingElement := FALSE;

            expectedTreeOutput1[19].types := SINT#16#0;
            expectedTreeOutput1[19].key := 'author';
            expectedTreeOutput1[19].value := 'J.K. Rowling';
            expectedTreeOutput1[19].depth := SINT#16#03;
            expectedTreeOutput1[19].closingElement := FALSE;

            expectedTreeOutput1[20].types := SINT#16#0;
            expectedTreeOutput1[20].key := 'year';
            expectedTreeOutput1[20].value := '1997';
            expectedTreeOutput1[20].depth := SINT#16#03;
            expectedTreeOutput1[20].closingElement := false;

            expectedTreeOutput1[21].types := SINT#16#0;
            expectedTreeOutput1[21].key := 'price';
            expectedTreeOutput1[21].value := '20.00';
            expectedTreeOutput1[21].depth := SINT#16#03;
            expectedTreeOutput1[21].closingElement := false;

            //Test2 Setup

            expectedTreeOutput2[0].types := SINT#16#0;
            expectedTreeOutput2[0].key := 'bookstore';
            expectedTreeOutput2[0].value := 'NULL';
            expectedTreeOutput2[0].depth := SINT#16#01;
            expectedTreeOutput2[0].closingElement := FALSE;

            expectedTreeOutput2[1].types := SINT#16#0;
            expectedTreeOutput2[1].key := 'book';
            expectedTreeOutput2[1].value := 'NULL';
            expectedTreeOutput2[1].depth := SINT#16#02;
            expectedTreeOutput2[1].closingElement := FALSE;

            expectedTreeOutput2[2].types := SINT#16#01;
            expectedTreeOutput2[2].key := 'category';
            expectedTreeOutput2[2].value := 'Science Fiction';
            expectedTreeOutput2[2].depth := SINT#16#02;
            expectedTreeOutput2[2].closingElement := FALSE;

            expectedTreeOutput2[3].types := SINT#16#01;
            expectedTreeOutput2[3].key := 'lang';
            expectedTreeOutput2[3].value := 'en';
            expectedTreeOutput2[3].depth := SINT#16#02;
            expectedTreeOutput2[3].closingElement := FALSE;

            expectedTreeOutput2[4].types := SINT#16#0;
            expectedTreeOutput2[4].key := 'title';
            expectedTreeOutput2[4].value := 'The Great Gatsby';
            expectedTreeOutput2[4].depth := SINT#16#03;
            expectedTreeOutput2[4].closingElement := FALSE;

            expectedTreeOutput2[5].types := SINT#16#0;
            expectedTreeOutput2[5].key := 'author';
            expectedTreeOutput2[5].value := 'F. Scott Fitzgerald';
            expectedTreeOutput2[5].depth := SINT#16#03;
            expectedTreeOutput2[5].closingElement := FALSE;

            expectedTreeOutput2[6].types := SINT#16#0;
            expectedTreeOutput2[6].key := 'year';
            expectedTreeOutput2[6].value := '1925';
            expectedTreeOutput2[6].depth := SINT#16#03;
            expectedTreeOutput2[6].closingElement := FALSE;

            expectedTreeOutput2[7].types := SINT#16#0;
            expectedTreeOutput2[7].key := 'price';
            expectedTreeOutput2[7].value := '10.99';
            expectedTreeOutput2[7].depth := SINT#16#03;
            expectedTreeOutput2[7].closingElement := FALSE;
        END_METHOD

        //Test1
        {Test}
        METHOD PUBLIC TestXmlDeserializer
            VAR
                i : INT;
            END_VAR;
            // Disable timeout timer for the test
            AxUnit.Mocking.Mock(mockeeFn := NAME_OF(System.Timer.OnDelay), mockFn := NAME_OF(Simatic.Ax.Mocks.OnDelayMock_false));

            xmlDeserializer.search := FALSE;
            xmlDeserializer.execute := TRUE;
            StringToByteArray(string1 := rawInput1, string2 := rawInput2, string3 := rawInput3, byteArray := rawInput);
            WHILE (TRUE) DO
                xmlDeserializer(raw := rawInput, tree := actualTreeOutput);
                // Copy data from the fixed-size byte array to xmlDeserializer.raw
                IF(xmlDeserializer.done = TRUE) THEN
                    EXIT;
                END_IF;
                IF(xmlDeserializer.error = TRUE) THEN
                    EXIT;
                END_IF;
            END_WHILE;
            //Test Block execution
            AxUnit.Assert.Equal(actual := xmlDeserializer.resultCount, expected := 22); //19
            AXUnit.Assert.Equal(actual := xmlDeserializer.busy, expected := FALSE);
            AXUnit.Assert.Equal(actual := xmlDeserializer.error, expected := FALSE);
            AXUnit.Assert.Equal(actual := xmlDeserializer.done, expected := TRUE);
            //Test Block Content
            Assert.LStreamTypeElementEqual(actualTreeOutput,expectedTreeOutput1);
        END_METHOD

        //Test2
        {Test}
        METHOD PUBLIC TestXmlDeserializer_Empty_Spaces
            // Disable timeout timer for the test
            AxUnit.Mocking.Mock(mockeeFn := NAME_OF(System.Timer.OnDelay), mockFn := NAME_OF(Simatic.Ax.Mocks.OnDelayMock_false));

            xmlDeserializer2.search := FALSE;
            xmlDeserializer2.execute := TRUE;

            StringToByteArray(string1 := rawInput4, byteArray := rawInput_2);

            WHILE (TRUE) DO
                xmlDeserializer2(raw := rawInput_2, tree := actualTreeOutput2);
                IF (xmlDeserializer2.done = TRUE) THEN
                    EXIT;
                END_IF;
                IF (xmlDeserializer2.error = TRUE) THEN
                    EXIT;
                END_IF;
            END_WHILE;

            AxUnit.Assert.Equal(actual := xmlDeserializer2.resultCount, expected := 8);
            AxUnit.Assert.Equal(actual := xmlDeserializer2.busy, expected := FALSE);
            AxUnit.Assert.Equal(actual := xmlDeserializer2.error, expected := FALSE);
            AxUnit.Assert.Equal(actual := xmlDeserializer2.done, expected := TRUE);
            Assert.LStreamTypeElementEqual(actualTreeOutput2, expectedTreeOutput2);
        END_METHOD
    END_CLASS
END_NAMESPACE

(* ---- XmlSerializerTests.st ---- *)
USING Simatic;
USING AxUnit;
USING Simatic.Ax.LStream;
USING Simatic.Ax.LStream.Utilities;
USING System.Strings;
USING Simatic.Ax.LStream.Models;

NAMESPACE LStreamTest
    ///////////////// Tests for XML Blocks
{TestFixture}
CLASS XmlSerializerTests
    VAR

        //Test1 (Test to try the LStream_XmlSerializer.st by serializing a tree (treeInput) and comparing its output (actualXmlByteArrayOutput) with the expected byte array (expectedXmlByteOutputResult))
        xmlSerializer : LStream_XmlSerializer;
        treeInput : ARRAY[0..200] OF LStream_typeElement;
        actualXmlByteArrayOutput : ARRAY[0..700] OF BYTE;
        expectedXmlByteOutputResult : ARRAY[0..507] OF BYTE := [
    BYTE#16#3C, BYTE#16#3F, BYTE#16#78, BYTE#16#6D, BYTE#16#6C, BYTE#16#20, BYTE#16#76, BYTE#16#65, BYTE#16#72, BYTE#16#73, BYTE#16#69, BYTE#16#6F,
    BYTE#16#6E, BYTE#16#3D, BYTE#16#22, BYTE#16#31, BYTE#16#2E, BYTE#16#30, BYTE#16#22, BYTE#16#20, BYTE#16#65, BYTE#16#6E, BYTE#16#63, BYTE#16#6F,
    BYTE#16#64, BYTE#16#69, BYTE#16#6E, BYTE#16#67, BYTE#16#3D, BYTE#16#22, BYTE#16#41, BYTE#16#53, BYTE#16#43, BYTE#16#49, BYTE#16#49, BYTE#16#22,
    BYTE#16#3F, BYTE#16#3E, BYTE#16#3C, BYTE#16#62, BYTE#16#6F, BYTE#16#6F, BYTE#16#6B, BYTE#16#73, BYTE#16#74, BYTE#16#6F, BYTE#16#72, BYTE#16#65,
    BYTE#16#3E, BYTE#16#3C, BYTE#16#62, BYTE#16#6F, BYTE#16#6F, BYTE#16#6B, BYTE#16#20, BYTE#16#63, BYTE#16#61, BYTE#16#74, BYTE#16#65, BYTE#16#67,
    BYTE#16#6F, BYTE#16#72, BYTE#16#79, BYTE#16#3D, BYTE#16#22, BYTE#16#46, BYTE#16#69, BYTE#16#63, BYTE#16#74, BYTE#16#69, BYTE#16#6F, BYTE#16#6E,
    BYTE#16#22, BYTE#16#3E, BYTE#16#3C, BYTE#16#74, BYTE#16#69, BYTE#16#74, BYTE#16#6C, BYTE#16#65, BYTE#16#20, BYTE#16#6C, BYTE#16#61, BYTE#16#6E,
    BYTE#16#67, BYTE#16#3D, BYTE#16#22, BYTE#16#65, BYTE#16#6E, BYTE#16#22, BYTE#16#3E, BYTE#16#54, BYTE#16#68, BYTE#16#65, BYTE#16#20, BYTE#16#47,
    BYTE#16#72, BYTE#16#65, BYTE#16#61, BYTE#16#74, BYTE#16#20, BYTE#16#47, BYTE#16#61, BYTE#16#74, BYTE#16#73, BYTE#16#62, BYTE#16#79, BYTE#16#3C,
    BYTE#16#2F, BYTE#16#74, BYTE#16#69, BYTE#16#74, BYTE#16#6C, BYTE#16#65, BYTE#16#3E, BYTE#16#3C, BYTE#16#61, BYTE#16#75, BYTE#16#74, BYTE#16#68,
    BYTE#16#6F, BYTE#16#72, BYTE#16#3E, BYTE#16#46, BYTE#16#2E, BYTE#16#20, BYTE#16#53, BYTE#16#63, BYTE#16#6F, BYTE#16#74, BYTE#16#74, BYTE#16#20,
    BYTE#16#46, BYTE#16#69, BYTE#16#74, BYTE#16#7A, BYTE#16#67, BYTE#16#65, BYTE#16#72, BYTE#16#61, BYTE#16#6C, BYTE#16#64, BYTE#16#3C, BYTE#16#2F,
    BYTE#16#61, BYTE#16#75, BYTE#16#74, BYTE#16#68, BYTE#16#6F, BYTE#16#72, BYTE#16#3E, BYTE#16#3C, BYTE#16#79, BYTE#16#65, BYTE#16#61, BYTE#16#72,
    BYTE#16#3E, BYTE#16#31, BYTE#16#39, BYTE#16#32, BYTE#16#35, BYTE#16#3C, BYTE#16#2F, BYTE#16#79, BYTE#16#65, BYTE#16#61, BYTE#16#72, BYTE#16#3E,
    BYTE#16#3C, BYTE#16#70, BYTE#16#72, BYTE#16#69, BYTE#16#63, BYTE#16#65, BYTE#16#3E, BYTE#16#31, BYTE#16#30, BYTE#16#2E, BYTE#16#39, BYTE#16#39,
    BYTE#16#3C, BYTE#16#2F, BYTE#16#70, BYTE#16#72, BYTE#16#69, BYTE#16#63, BYTE#16#65, BYTE#16#3E, BYTE#16#3C, BYTE#16#2F, BYTE#16#62, BYTE#16#6F,
    BYTE#16#6F, BYTE#16#6B, BYTE#16#3E, BYTE#16#3C, BYTE#16#62, BYTE#16#6F, BYTE#16#6F, BYTE#16#6B, BYTE#16#20, BYTE#16#63, BYTE#16#61, BYTE#16#74,
    BYTE#16#65, BYTE#16#67, BYTE#16#6F, BYTE#16#72, BYTE#16#79, BYTE#16#3D, BYTE#16#22, BYTE#16#50, BYTE#16#72, BYTE#16#6F, BYTE#16#67, BYTE#16#72,
    BYTE#16#61, BYTE#16#6D, BYTE#16#6D, BYTE#16#69, BYTE#16#6E, BYTE#16#67, BYTE#16#22, BYTE#16#3E, BYTE#16#3C, BYTE#16#74, BYTE#16#69, BYTE#16#74,
    BYTE#16#6C, BYTE#16#65, BYTE#16#20, BYTE#16#6C, BYTE#16#61, BYTE#16#6E, BYTE#16#67, BYTE#16#3D, BYTE#16#22, BYTE#16#65, BYTE#16#6E, BYTE#16#22,
    BYTE#16#3E, BYTE#16#4C, BYTE#16#65, BYTE#16#61, BYTE#16#72, BYTE#16#6E, BYTE#16#69, BYTE#16#6E, BYTE#16#67, BYTE#16#20, BYTE#16#58, BYTE#16#4D,
    BYTE#16#4C, BYTE#16#3C, BYTE#16#2F, BYTE#16#74, BYTE#16#69, BYTE#16#74, BYTE#16#6C, BYTE#16#65, BYTE#16#3E, BYTE#16#3C, BYTE#16#61, BYTE#16#75,
    BYTE#16#74, BYTE#16#68, BYTE#16#6F, BYTE#16#72, BYTE#16#3E, BYTE#16#45, BYTE#16#72, BYTE#16#69, BYTE#16#6B, BYTE#16#20, BYTE#16#54, BYTE#16#2E,
    BYTE#16#20, BYTE#16#52, BYTE#16#61, BYTE#16#79, BYTE#16#3C, BYTE#16#2F, BYTE#16#61, BYTE#16#75, BYTE#16#74, BYTE#16#68, BYTE#16#6F, BYTE#16#72,
    BYTE#16#3E, BYTE#16#3C, BYTE#16#79, BYTE#16#65, BYTE#16#61, BYTE#16#72, BYTE#16#3E, BYTE#16#32, BYTE#16#30, BYTE#16#30, BYTE#16#33, BYTE#16#3C,
    BYTE#16#2F, BYTE#16#79, BYTE#16#65, BYTE#16#61, BYTE#16#72, BYTE#16#3E, BYTE#16#3C, BYTE#16#70, BYTE#16#72, BYTE#16#69, BYTE#16#63, BYTE#16#65,
    BYTE#16#3E, BYTE#16#33, BYTE#16#39, BYTE#16#2E, BYTE#16#39, BYTE#16#35, BYTE#16#3C, BYTE#16#2F, BYTE#16#70, BYTE#16#72, BYTE#16#69, BYTE#16#63,
    BYTE#16#65, BYTE#16#3E, BYTE#16#3C, BYTE#16#2F, BYTE#16#62, BYTE#16#6F, BYTE#16#6F, BYTE#16#6B, BYTE#16#3E, BYTE#16#3C, BYTE#16#62, BYTE#16#6F,
    BYTE#16#6F, BYTE#16#6B, BYTE#16#20, BYTE#16#63, BYTE#16#61, BYTE#16#74, BYTE#16#65, BYTE#16#67, BYTE#16#6F, BYTE#16#72, BYTE#16#79, BYTE#16#3D,
    BYTE#16#22, BYTE#16#46, BYTE#16#61, BYTE#16#6E, BYTE#16#74, BYTE#16#61, BYTE#16#73, BYTE#16#79, BYTE#16#22, BYTE#16#3E, BYTE#16#3C, BYTE#16#74,
    BYTE#16#69, BYTE#16#74, BYTE#16#6C, BYTE#16#65, BYTE#16#20, BYTE#16#6C, BYTE#16#61, BYTE#16#6E, BYTE#16#67, BYTE#16#3D, BYTE#16#22, BYTE#16#65,
    BYTE#16#6E, BYTE#16#22, BYTE#16#3E, BYTE#16#48, BYTE#16#61, BYTE#16#72, BYTE#16#72, BYTE#16#79, BYTE#16#20, BYTE#16#50, BYTE#16#6F, BYTE#16#74,
    BYTE#16#74, BYTE#16#65, BYTE#16#72, BYTE#16#20, BYTE#16#61, BYTE#16#6E, BYTE#16#64, BYTE#16#20, BYTE#16#74, BYTE#16#68, BYTE#16#65, BYTE#16#20,
    BYTE#16#50, BYTE#16#68, BYTE#16#69, BYTE#16#6C, BYTE#16#6F, BYTE#16#73, BYTE#16#6F, BYTE#16#70, BYTE#16#68, BYTE#16#65, BYTE#16#72, BYTE#16#73,
    BYTE#16#20, BYTE#16#53, BYTE#16#74, BYTE#16#6F, BYTE#16#6E, BYTE#16#65, BYTE#16#3C, BYTE#16#2F, BYTE#16#74, BYTE#16#69, BYTE#16#74, BYTE#16#6C,
    BYTE#16#65, BYTE#16#3E, BYTE#16#3C, BYTE#16#61, BYTE#16#75, BYTE#16#74, BYTE#16#68, BYTE#16#6F, BYTE#16#72, BYTE#16#3E, BYTE#16#4A, BYTE#16#2E,
    BYTE#16#4B, BYTE#16#2E, BYTE#16#20, BYTE#16#52, BYTE#16#6F, BYTE#16#77, BYTE#16#6C, BYTE#16#69, BYTE#16#6E, BYTE#16#67, BYTE#16#3C, BYTE#16#2F,
    BYTE#16#61, BYTE#16#75, BYTE#16#74, BYTE#16#68, BYTE#16#6F, BYTE#16#72, BYTE#16#3E, BYTE#16#3C, BYTE#16#79, BYTE#16#65, BYTE#16#61, BYTE#16#72,
    BYTE#16#3E, BYTE#16#31, BYTE#16#39, BYTE#16#39, BYTE#16#37, BYTE#16#3C, BYTE#16#2F, BYTE#16#79, BYTE#16#65, BYTE#16#61, BYTE#16#72, BYTE#16#3E,
    BYTE#16#3C, BYTE#16#70, BYTE#16#72, BYTE#16#69, BYTE#16#63, BYTE#16#65, BYTE#16#3E, BYTE#16#32, BYTE#16#30, BYTE#16#2E, BYTE#16#30, BYTE#16#30,
    BYTE#16#3C, BYTE#16#2F, BYTE#16#70, BYTE#16#72, BYTE#16#69, BYTE#16#63, BYTE#16#65, BYTE#16#3E, BYTE#16#3C, BYTE#16#2F, BYTE#16#62, BYTE#16#6F,
    BYTE#16#6F, BYTE#16#6B, BYTE#16#3E, BYTE#16#3C, BYTE#16#2F, BYTE#16#62, BYTE#16#6F, BYTE#16#6F, BYTE#16#6B, BYTE#16#73, BYTE#16#74, BYTE#16#6F,
    BYTE#16#72, BYTE#16#65, BYTE#16#3E, BYTE#16#0];

       // Test 2 (Test to try the LStream_XmlSerializer.st when the input tree (treeInput2) contains empty nodes (either 'NULL' or ''). In this example, the empty nodes are treeInput2[5] and treeInput2[7])
        xmlSerializer2 : LStream_XmlSerializer;
        treeInput2 : ARRAY[0..200] OF LStream_typeElement;
        actualXmlByteArrayOutput2 : ARRAY[0..700] OF BYTE;
        expectedXmlByteOutputResult2 : ARRAY[0..170] OF BYTE := [
    BYTE#16#3C, BYTE#16#3F, BYTE#16#78, BYTE#16#6D, BYTE#16#6C, BYTE#16#20, BYTE#16#76, BYTE#16#65, BYTE#16#72, BYTE#16#73, BYTE#16#69, BYTE#16#6F, BYTE#16#6E, BYTE#16#3D, BYTE#16#22, BYTE#16#31,
    BYTE#16#2E, BYTE#16#30, BYTE#16#22, BYTE#16#20, BYTE#16#65, BYTE#16#6E, BYTE#16#63, BYTE#16#6F, BYTE#16#64, BYTE#16#69, BYTE#16#6E, BYTE#16#67, BYTE#16#3D, BYTE#16#22, BYTE#16#41, BYTE#16#53,
    BYTE#16#43, BYTE#16#49, BYTE#16#49, BYTE#16#22, BYTE#16#3F, BYTE#16#3E, BYTE#16#3C, BYTE#16#62, BYTE#16#6F, BYTE#16#6F, BYTE#16#6B, BYTE#16#73, BYTE#16#74, BYTE#16#6F, BYTE#16#72, BYTE#16#65,
    BYTE#16#3E, BYTE#16#3C, BYTE#16#62, BYTE#16#6F, BYTE#16#6F, BYTE#16#6B, BYTE#16#20, BYTE#16#63, BYTE#16#61, BYTE#16#74, BYTE#16#65, BYTE#16#67, BYTE#16#6F, BYTE#16#72, BYTE#16#79, BYTE#16#3D,
    BYTE#16#22, BYTE#16#46, BYTE#16#69, BYTE#16#63, BYTE#16#74, BYTE#16#69, BYTE#16#6F, BYTE#16#6E, BYTE#16#22, BYTE#16#3E, BYTE#16#3C, BYTE#16#74, BYTE#16#69, BYTE#16#74, BYTE#16#6C, BYTE#16#65,
    BYTE#16#20, BYTE#16#6C, BYTE#16#61, BYTE#16#6E, BYTE#16#67, BYTE#16#3D, BYTE#16#22, BYTE#16#65, BYTE#16#6E, BYTE#16#22, BYTE#16#3E, BYTE#16#4A, BYTE#16#61, BYTE#16#77, BYTE#16#73, BYTE#16#3C,
    BYTE#16#2F, BYTE#16#74, BYTE#16#69, BYTE#16#74, BYTE#16#6C, BYTE#16#65, BYTE#16#3E, BYTE#16#3C, BYTE#16#61, BYTE#16#75, BYTE#16#74, BYTE#16#68, BYTE#16#6F, BYTE#16#72, BYTE#16#3E, BYTE#16#3C,
    BYTE#16#2F, BYTE#16#61, BYTE#16#75, BYTE#16#74, BYTE#16#68, BYTE#16#6F, BYTE#16#72, BYTE#16#3E, BYTE#16#3C, BYTE#16#79, BYTE#16#65, BYTE#16#61, BYTE#16#72, BYTE#16#3E, BYTE#16#32, BYTE#16#30,
    BYTE#16#30, BYTE#16#31, BYTE#16#3C, BYTE#16#2F, BYTE#16#79, BYTE#16#65, BYTE#16#61, BYTE#16#72, BYTE#16#3E, BYTE#16#3C, BYTE#16#70, BYTE#16#72, BYTE#16#69, BYTE#16#63, BYTE#16#65, BYTE#16#3E,
    BYTE#16#3C, BYTE#16#2F, BYTE#16#70, BYTE#16#72, BYTE#16#69, BYTE#16#63, BYTE#16#65, BYTE#16#3E, BYTE#16#3C, BYTE#16#2F, BYTE#16#62, BYTE#16#6F, BYTE#16#6F, BYTE#16#6B, BYTE#16#3E, BYTE#16#3C,
    BYTE#16#2F, BYTE#16#62, BYTE#16#6F, BYTE#16#6F, BYTE#16#6B, BYTE#16#73, BYTE#16#74, BYTE#16#6F, BYTE#16#72, BYTE#16#65, BYTE#16#3E];
    END_VAR

    {FixtureSetup}
    METHOD PUBLIC TestSetup
        //Populate tree input
        treeInput[0].types := SINT#16#0;
        treeInput[0].key := 'bookstore';
        treeInput[0].value := 'NULL';
        treeInput[0].depth := SINT#16#01;
        treeInput[0].closingElement := FALSE;

        treeInput[1].types := SINT#16#0;
        treeInput[1].key := 'book';
        treeInput[1].value := 'NULL';
        treeInput[1].depth := SINT#16#02;
        treeInput[1].closingElement := FALSE;

        treeInput[2].types := SINT#16#01;
        treeInput[2].key := 'category';
        treeInput[2].value := 'Fiction';
        treeInput[2].depth := SINT#16#02;
        treeInput[2].closingElement := FALSE;

        treeInput[3].types := SINT#16#0;
        treeInput[3].key := 'title';
        treeInput[3].value := 'The Great Gatsby';
        treeInput[3].depth := SINT#16#03;
        treeInput[3].closingElement := FALSE;

        treeInput[4].types := SINT#16#01;
        treeInput[4].key := 'lang';
        treeInput[4].value := 'en';
        treeInput[4].depth := SINT#16#03;
        treeInput[4].closingElement := FALSE;

        treeInput[5].types := SINT#16#0;
        treeInput[5].key := 'author';
        treeInput[5].value := 'F. Scott Fitzgerald';
        treeInput[5].depth := SINT#16#03;
        treeInput[5].closingElement := false;

        treeInput[6].types := SINT#16#0;
        treeInput[6].key := 'year';
        treeInput[6].value := '1925';
        treeInput[6].depth := SINT#16#03;
        treeInput[6].closingElement := false;

        treeInput[7].types := SINT#16#0;
        treeInput[7].key := 'price';
        treeInput[7].value := '10.99';
        treeInput[7].depth := SINT#16#03;
        treeInput[7].closingElement := false;

        treeInput[8].types := SINT#16#0;
        treeInput[8].key := 'book';
        treeInput[8].value := 'NULL';
        treeInput[8].depth := SINT#16#02;
        treeInput[8].closingElement := false;

        treeInput[9].types := SINT#16#01;
        treeInput[9].key := 'category';
        treeInput[9].value := 'Programming';
        treeInput[9].depth := SINT#16#02;
        treeInput[9].closingElement := false;

        treeInput[10].types := SINT#16#0;
        treeInput[10].key := 'title';
        treeInput[10].value := 'Learning XML';
        treeInput[10].depth := SINT#16#03;
        treeInput[10].closingElement := false;

        treeInput[11].types := SINT#16#01;
        treeInput[11].key := 'lang';
        treeInput[11].value := 'en';
        treeInput[11].depth := SINT#16#03;
        treeInput[11].closingElement := FALSE;

        treeInput[12].types := SINT#16#0;
        treeInput[12].key := 'author';
        treeInput[12].value := 'Erik T. Ray';
        treeInput[12].depth := SINT#16#03;
        treeInput[12].closingElement := false;

        treeInput[13].types := SINT#16#0;
        treeInput[13].key := 'year';
        treeInput[13].value := '2003';
        treeInput[13].depth := SINT#16#03;
        treeInput[13].closingElement := false;

        treeInput[14].types := SINT#16#0;
        treeInput[14].key := 'price';
        treeInput[14].value := '39.95';
        treeInput[14].depth := SINT#16#03;
        treeInput[14].closingElement := false;

        treeInput[15].types := SINT#16#0;
        treeInput[15].key := 'book';
        treeInput[15].value := 'NULL';
        treeInput[15].depth := SINT#16#02;
        treeInput[15].closingElement := false;

        treeInput[16].types := SINT#16#01;
        treeInput[16].key := 'category';
        treeInput[16].value := 'Fantasy';
        treeInput[16].depth := SINT#16#02;
        treeInput[16].closingElement := FALSE;

        treeInput[17].types := SINT#16#0;
        treeInput[17].key := 'title';
        treeInput[17].value := 'Harry Potter and the Philosophers Stone';
        treeInput[17].depth := SINT#16#03;
        treeInput[17].closingElement := FALSE;

        treeInput[18].types := SINT#16#01;
        treeInput[18].key := 'lang';
        treeInput[18].value := 'en';
        treeInput[18].depth := SINT#16#03;
        treeInput[18].closingElement := FALSE;

        treeInput[19].types := SINT#16#0;
        treeInput[19].key := 'author';
        treeInput[19].value := 'J.K. Rowling';
        treeInput[19].depth := SINT#16#03;
        treeInput[19].closingElement := FALSE;

        treeInput[20].types := SINT#16#0;
        treeInput[20].key := 'year';
        treeInput[20].value := '1997';
        treeInput[20].depth := SINT#16#03;
        treeInput[20].closingElement := false;

        treeInput[21].types := SINT#16#0;
        treeInput[21].key := 'price';
        treeInput[21].value := '20.00';
        treeInput[21].depth := SINT#16#03;
        treeInput[21].closingElement := false;

        //Test2 Setup
        treeInput2[0].types := SINT#16#0;
        treeInput2[0].key := 'bookstore';
        treeInput2[0].value := 'NULL';
        treeInput2[0].depth := SINT#16#01;
        treeInput2[0].closingElement := FALSE;

        treeInput2[1].types := SINT#16#0;
        treeInput2[1].key := 'book';
        treeInput2[1].value := 'NULL';
        treeInput2[1].depth := SINT#16#02;
        treeInput2[1].closingElement := FALSE;

        treeInput2[2].types := SINT#16#01;
        treeInput2[2].key := 'category';
        treeInput2[2].value := 'Fiction';
        treeInput2[2].depth := SINT#16#02;
        treeInput2[2].closingElement := FALSE;

        treeInput2[3].types := SINT#16#0;
        treeInput2[3].key := 'title';
        treeInput2[3].value := 'Jaws';
        treeInput2[3].depth := SINT#16#03;
        treeInput2[3].closingElement := FALSE;

        treeInput2[4].types := SINT#16#01;
        treeInput2[4].key := 'lang';
        treeInput2[4].value := 'en';
        treeInput2[4].depth := SINT#16#03;
        treeInput2[4].closingElement := FALSE;

        treeInput2[5].types := SINT#16#0;
        treeInput2[5].key := 'author';
        treeInput2[5].value := 'NULL';
        treeInput2[5].depth := SINT#16#03;
        treeInput2[5].closingElement := FALSE;

        treeInput2[6].types := SINT#16#0;
        treeInput2[6].key := 'year';
        treeInput2[6].value := '2001';
        treeInput2[6].depth := SINT#16#03;
        treeInput2[6].closingElement := FALSE;

        treeInput2[7].types := SINT#16#0;
        treeInput2[7].key := 'price';
        treeInput2[7].value := '';
        treeInput2[7].depth := SINT#16#03;
        treeInput2[7].closingElement := FALSE;

    END_METHOD

    {Test}
    METHOD PUBLIC TestXmlSerializer
        VAR
            i : INT;
        END_VAR;
        // Disable timeout timer for the test
        AxUnit.Mocking.Mock(mockeeFn := NAME_OF(System.Timer.OnDelay), mockFn := NAME_OF(Simatic.Ax.Mocks.OnDelayMock_false));

        xmlSerializer.execute := TRUE;
        WHILE (i < 200) DO
            xmlSerializer(tree := treeInput, xmlByteArray := actualXmlByteArrayOutput);
            IF(xmlSerializer.done = TRUE) THEN
                EXIT;
            END_IF;
            IF(xmlSerializer.error = TRUE) THEN
                EXIT;
            END_IF;
            i := i +1;
        END_WHILE;

        //Test Block execution
        AxUnit.Assert.Equal(actual := xmlSerializer.count, expected := UINT#507); //19
        AXUnit.Assert.Equal(actual := xmlSerializer.busy, expected := FALSE);
        AXUnit.Assert.Equal(actual := xmlSerializer.error, expected := FALSE);
        AXUnit.Assert.Equal(actual := xmlSerializer.done, expected := TRUE);

         //Test Content

        //Test Output Content
        FOR i := 0 TO 507 DO
            AxUnit.Assert.Equal(actualXmlByteArrayOutput[i], expectedXmlByteOutputResult[i]);
        END_FOR;

    END_METHOD

    {Test}
    METHOD PUBLIC TestXmlSerializer_EmptyValueNodes
        VAR
            i : INT;
        END_VAR;
        // Disable timeout timer for the test
        AxUnit.Mocking.Mock(mockeeFn := NAME_OF(System.Timer.OnDelay), mockFn := NAME_OF(Simatic.Ax.Mocks.OnDelayMock_false));

        xmlSerializer2.execute := TRUE;

        WHILE (i < 200) DO
            xmlSerializer2(tree := treeInput2, xmlByteArray := actualXmlByteArrayOutput2);
            IF(xmlSerializer2.done = TRUE) THEN
                EXIT;
            END_IF;
            IF(xmlSerializer2.error = TRUE) THEN
                EXIT;
            END_IF;
            i := i + 1;
        END_WHILE;

        //Test Block execution
        AxUnit.Assert.Equal(actual := xmlSerializer2.count, expected := UINT#171);
        AXUnit.Assert.Equal(actual := xmlSerializer2.busy, expected := FALSE);
        AXUnit.Assert.Equal(actual := xmlSerializer2.error, expected := FALSE);
        AXUnit.Assert.Equal(actual := xmlSerializer2.done, expected := TRUE);

         //Test Content

         //Test Output Content
        FOR i := 0 TO 170 DO
            AxUnit.Assert.Equal(actualXmlByteArrayOutput2[i], expectedXmlByteOutputResult2[i]);
        END_FOR;
    END_METHOD

END_CLASS
END_NAMESPACE
